{attribute 'OPC.UA.DA' := '0'}
TYPE IonizerAlarm :
STRUCT
	Name : STRING;
	Description : STRING;
	AlarmID : UINT;
	Triggered AT %I* : BOOL;
END_STRUCT
END_TYPE

(* stored: Version 1.1.0.1, ProductVersion 3.1.4024.12
   DUT IonizerAlarm: Id {51057726-62e4-43c5-84fe-a9b81c3bbe23} *)
